TYPE ST_FeedInToWareHouse_Status EXTENDS ST_StatusBasic :
STRUCT
END_STRUCT
END_TYPE

(* stored: Version 1.1.0.1, ProductVersion 3.1.4024.13
   DUT ST_FeedInToWareHouse_Status: Id {a1b2c3d4-6666-4aaa-b666-666666666602} *)
